// TIA Portal V19 export
TYPE "PosFbk_AnalogIn_Alr"
// stored: Access Published
   STRUCT
      CommFault : Bool;   // Communication fault
      SensorFault : Bool;   // Secnsor fault
      Resolution : Bool;   // Resolution is at 0
   END_STRUCT;
END_TYPE
